TYPE ST_SealerRecipe :
	STRUCT
		Axis		   : ST_AxisRecipe;
		Temp		   : LREAL := 100;
		SealTime	   : LREAL := 250;
		OpenPosition   : LREAL := 105;
		ClosedPosition : LREAL := 200;
	END_STRUCT
END_TYPE

(* stored: Version 1.1.0.1, ProductVersion 3.1.4026.18
   DUT ST_SealerRecipe: Id {5efbb8de-476a-442c-ac51-43f16c9d5a2a} *)
